FUNCTION_BLOCK FB_ProgressBar
VAR_INPUT
END_VAR
VAR_OUTPUT
END_VAR
VAR
END_VAR

END_FUNCTION_BLOCK

(* stored: Version 1.1.0.1
   POU FB_ProgressBar: Id {b42bd780-f298-0c3f-1cc9-ca2665c7b984}, SpecialFunc None *)
